// SIMATIC S7-200 project (STEP 7-Micro/WIN), CPU 215 REL 01.02

ORGANIZATION_BLOCK MAIN:OB1
TITLE=程序实现了木材加工厂中木片料仓的推料器系统。
// 系统的运行流程如下：
// 1.系统通过启动按钮启动运行，结合料仓空传感器的状态设置启动标志。
// 2.在自动模式下，推料器前进只能在启动标志为真，料仓满传感器未触发，推料器后退未激活，且推料器后退延时未超时的情况下激活，确保料仓未满时木片被推向加工设备。
// 3.推料器后退只能在料仓满传感器触发且启动标志为真，或料仓满标志为真的情况下激活，保证料仓满时推料器退回，避免过载。
// 4.系统支持手动操作，手动推料前进在手动推料按钮按下，手动推料后退未激活，或手动推料前进或料仓满标志为真，且推料器前进延时和手动推料前进延时超时，紧急停止标志和停止按钮未激活，启动标志为真的情况下激活，确保手动推送的安全性。
// 5.手动推料后退在停止按钮按下，或手动推料后退为真，手动推料前进未激活，且推料器前进延时和手动推料后退延时超时，紧急停止标志和手动推料按钮未激活，启动标志为真的情况下激活，保证手动退回的顺畅性。
// 6.手动推料标志在停止按钮未按下，手动推料按钮按下，手动推料前进和手动推料后退未激活，且紧急停止标志为假的情况下设置，明确手动模式的优先级。
// 7.紧急停止按钮触发时，紧急停止标志在紧急停止按钮按下，或紧急停止标志为真，且紧急停止后延时超时，紧急停止延时未超时的情况下设置，确保系统在紧急情况下停止动作。
// 
// 
BEGIN
Network 1
LD     I0.0
LPS
AN     T39
=      M0.0
LPP
A      I0.5
TON    T39, +30
Network 2
LD     M0.0
AN     I0.4
AN     Q0.1
AN     T37
=      Q0.0
TON    T44, +120
Network 3
LD     I0.4
A      M0.0
O      M0.3
LPS
=      Q0.1
AN     I0.4
TON    T37, +50
LRD
A      I0.4
TON    T40, +20
LPP
AN     T37
=      M0.3
Network 4
LD     I0.2
AN     Q0.3
O      Q0.2
O      M0.3
A      T44
AN     M0.1
AN     I0.1
A      M0.0
LPS
A      T42
=      Q0.2
LPP
TON    T42, +60
Network 5
LD     I0.1
O      Q0.3
AN     Q0.2
A      T44
AN     M0.1
AN     I0.2
A      M0.0
LPS
A      T43
=      Q0.3
LPP
TON    T43, +1
Network 6
LD     I0.3
O      M0.1
LPS
A      T41
AN     T38
=      M0.1
LRD
AN     I0.3
TON    T38, +100
LPP
TON    T41, +20
Network 7
LDN    I0.1
AI     I0.2
AN     Q0.2
AN     Q0.3
AN     M0.1
=      M0.2
END_ORGANIZATION_BLOCK
